(* PLC project Unnamed, Unknown Unnamed 1 *)
(* stored: creationDateTime 2026-02-17T10:07:24, modificationDateTime 2026-02-17T10:07:24 *)

(* 17 Feb Practise Task *)
PROGRAM main
  VAR
    Output : BOOL;
  END_VAR

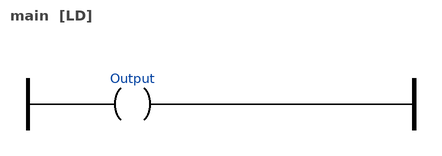
(* LD diagram, written out as Structured Text *)
Output := TRUE;
END_PROGRAM

CONFIGURATION Config0
  RESOURCE Res0 ON PLC
    TASK task0(INTERVAL := T#20ms, PRIORITY := 1);
    PROGRAM instance0 WITH task0 : main;
  END_RESOURCE
END_CONFIGURATION
